Staubli VAL3: writeENC.pgx

program writeENC()
  local bool l_bResult
  local num l_nError
  local num l_nValue
  local string l_sValue
begin
  // Update variables of the conveyor library
  resize(sCaption,1,pg:nNumOfTxtBox)
  call pg:getCaption(sCaption)
  //
  // LatchPeriod
  call pg:getFieldValue(sCaption[0],l_sValue,l_nError)
  toNum(l_sValue,enc:nLatchPeriod,l_bResult)
  // Encoder Resolution
  call pg:getFieldValue(sCaption[1],l_sValue,l_nError)
  toNum(l_sValue,cnv:nENCRESOLUTION,l_bResult)
  call enc:setResolution(cnv:nENCRESOLUTION)
  // FIR filter length
  call pg:getFieldValue(sCaption[2],l_sValue,l_nError)
  toNum(l_sValue,cnv:nFirOrdre,l_bResult)
  // FIR filter Delay
  call pg:getFieldValue(sCaption[3],l_sValue,l_nError)
  toNum(l_sValue,l_nValue,l_bResult)
  cnv:nFirDelay=l_nValue/1000
end
